// TIA Portal project "LinkedList_v000_000_004" (V16)
// task for 000.000.004: create LinkedList.FindID

(* hardware
DEVICE "S7-1200 station_1"  S7-1200 Station
   slot 0: "Rack_0"  S7-1200 Rack  Rack  V1.0
   slot 1: "PLC_1"  CPU 1212C DC/DC/DC  6ES7 212-1AE40-0XB0  V4.4
*)

// ===== PLC "PLC_1"  CPU 1212C DC/DC/DC =====

VAR_GLOBAL   // PLC tag table "Default tag table"
   "System_Byte" AT %MB1 : Byte;
   "FirstScan" AT %M1.0 : Bool;
   "DiagStatusUpdate" AT %M1.1 : Bool;
   "AlwaysTRUE" AT %M1.2 : Bool;
   "AlwaysFALSE" AT %M1.3 : Bool;
   "Clock_Byte" AT %MB0 : Byte;
   "Clock_10Hz" AT %M0.0 : Bool;
   "Clock_5Hz" AT %M0.1 : Bool;
   "Clock_2.5Hz" AT %M0.2 : Bool;
   "Clock_2Hz" AT %M0.3 : Bool;
   "Clock_1.25Hz" AT %M0.4 : Bool;
   "Clock_1Hz" AT %M0.5 : Bool;
   "Clock_0.625Hz" AT %M0.6 : Bool;
   "Clock_0.5Hz" AT %M0.7 : Bool;
END_VAR

TYPE "LinkedList.Node.Payload.UDT"
   STRUCT
      id : Char;
      status : String;
   END_STRUCT;
END_TYPE

TYPE "LinkedList.Node.UDT"
   STRUCT
      payload : "LinkedList.Node.Payload.UDT";
      pointer : DInt;
   END_STRUCT;
END_TYPE

TYPE "LinkedList.UDT"
   STRUCT
      head : DInt;
      list : Array[0..4] of "LinkedList.Node.UDT";
   END_STRUCT;
END_TYPE

TYPE "Validate.LinkedList.FindPointer.UDT"
   STRUCT
      request : Bool;
      needle : DInt;
      not_found : DInt;
      index : DInt;
   END_STRUCT;
END_TYPE

TYPE "Validate.LinkedList.FindPayload.UDT"
   STRUCT
      request : Bool;
      needle : "LinkedList.Node.Payload.UDT";
      not_found : DInt;
      tail_address : DInt;
      index : DInt;
   END_STRUCT;
END_TYPE

TYPE "Validate.LinkedList.FindID.UDT"
   STRUCT
      request : Bool;
      needle : Char;
      not_found : DInt;
      tail_address : DInt;
      index : DInt;
   END_STRUCT;
END_TYPE

DATA_BLOCK "LinkedList.IDB"   // DB1
{ S7_Optimized_Access := 'TRUE' }
AUTHOR : Machado
FAMILY : LinkedList
VERSION : 0.1
// stored: InstanceOfName LinkedList
"LinkedList"
BEGIN
END_DATA_BLOCK

DATA_BLOCK "ValidationSignals"   // DB2
{ S7_Optimized_Access := 'TRUE' }
VERSION : 0.1
   VAR
      FindPointer : "Validate.LinkedList.FindPointer.UDT";
      FindPayload : "Validate.LinkedList.FindPayload.UDT";
      FindID : "Validate.LinkedList.FindID.UDT";
   END_VAR
BEGIN
END_DATA_BLOCK

FUNCTION_BLOCK "LinkedList"   // FB1, SCL
TITLE = Linked List
{ S7_Optimized_Access := 'TRUE' }
AUTHOR : Machado
FAMILY : LinkedList
VERSION : 0.1
   VAR
      list : "LinkedList.UDT";
   END_VAR
BEGIN
END_FUNCTION_BLOCK

FUNCTION "LinkedList.FindPointer" : DInt   // FC1, SCL
TITLE = Find Node by Pointer In Linked List
{ S7_Optimized_Access := 'TRUE' }
AUTHOR : Machado
FAMILY : LinkedList
VERSION : 0.1
// returns not_found when not found.
// otherwise returs index of parent array where node with needle value as pointer.
   VAR_INPUT
      needle : DInt;
      not_found : DInt;   // value returned to user if needle not found
   END_VAR
   VAR_IN_OUT
      haystack : "LinkedList.UDT";
   END_VAR
   VAR_TEMP
      i : DInt;
      size : DInt;
   END_VAR
BEGIN
   REGION "GET SIZE"
       #size := UDINT_TO_DINT("LinkedList.Node[].CountOfElements"(#haystack.list));
   END_REGION


   REGION "SEARCH"
       FOR #i := 0 TO #size - 1 DO
           // no match
           IF #haystack.list[#i]."pointer" <> #needle THEN
               CONTINUE;
           END_IF;
           // match
           #"LinkedList.FindPointer" := #i;
           RETURN;
       END_FOR;
   END_REGION


   REGION "NOT FOUND"
       #"LinkedList.FindPointer" := #not_found;
       RETURN;
   END_REGION
END_FUNCTION

FUNCTION "LinkedList.Node[].CountOfElements" : UDInt   // FC2, SCL
TITLE = Count Of Elements of an Array of Linked List Nodes
{ S7_Optimized_Access := 'TRUE' }
AUTHOR : Machado
FAMILY : LinkedList
VERSION : 0.1
   VAR_INPUT
      list : Variant;
   END_VAR
BEGIN
   #"LinkedList.Node[].CountOfElements" := CountOfElements(#list);
   RETURN;
END_FUNCTION

FUNCTION "LinkedList.FindPayload" : DInt   // FC3, SCL
TITLE = Finde Node Index By Payload
{ S7_Optimized_Access := 'TRUE' }
AUTHOR : Machado
FAMILY : LinkedList
VERSION : 0.1
   VAR_INPUT
      needle : "LinkedList.Node.Payload.UDT";
      not_found : DInt;
      tail_address : DInt;
   END_VAR
   VAR_IN_OUT
      haystack : "LinkedList.UDT";
   END_VAR
   VAR_TEMP
      size : DInt;
      this_node : "LinkedList.Node.UDT";
      next_node : "LinkedList.Node.UDT";
      nodes_visited : DInt;
   END_VAR
BEGIN
   REGION "GET SIZE"
       #size := UDINT_TO_DINT("LinkedList.Node[].CountOfElements"(#haystack.list));
   END_REGION


   REGION "PRE-CONDITIONS"
       IF NOT "DInt.InRange"(x := #haystack.head, max := #size - 1, min := 0) THEN
           #"LinkedList.FindPayload" := #not_found;
           RETURN;
       END_IF;
   END_REGION


   REGION "PRIME WHILE LOOP"
       #this_node := #haystack.list[#haystack.head];
       IF #this_node.payload = #needle THEN
           #"LinkedList.FindPayload" := #haystack.head;
           RETURN;
       END_IF;
       #nodes_visited := 1;
   END_REGION


   REGION "SEARCH"
       WHILE #this_node."pointer" <> #tail_address DO
           #next_node := #haystack.list[#this_node."pointer"];
           IF #next_node.payload = #needle THEN
               #"LinkedList.FindPayload" := #this_node."pointer";
               RETURN;
           END_IF;
           #nodes_visited += 1;
           IF #nodes_visited > #size THEN
               #"LinkedList.FindPayload" := #not_found;
               RETURN;
           END_IF;
           #this_node := #next_node;
       END_WHILE;
   END_REGION


   REGION "NOT FOUND"
       #"LinkedList.FindPayload" := #not_found;
       RETURN;
   END_REGION
END_FUNCTION

FUNCTION "DInt.InRange" : Bool   // FC4, SCL
TITLE = Value Is In Range
{ S7_Optimized_Access := 'TRUE' }
AUTHOR : Machado
FAMILY : DInt
VERSION : 0.1
   VAR_INPUT
      x : DInt;
      max : DInt;
      min : DInt;
   END_VAR
BEGIN
   #"DInt.InRange" := #min <= #x AND #x <= #max;
END_FUNCTION

FUNCTION "LinkedList.FindID" : DInt   // FC5, SCL
TITLE = Finde Node Index By Payload
{ S7_Optimized_Access := 'TRUE' }
AUTHOR : Machado
FAMILY : LinkedList
VERSION : 0.1
   VAR_INPUT
      needle : Char;
      not_found : DInt;
      tail_address : DInt;
   END_VAR
   VAR_IN_OUT
      haystack : "LinkedList.UDT";
   END_VAR
   VAR_TEMP
      size : DInt;
      this_node : "LinkedList.Node.UDT";
      next_node : "LinkedList.Node.UDT";
      nodes_visited : DInt;
   END_VAR
BEGIN
   REGION "GET SIZE"
       #size := UDINT_TO_DINT("LinkedList.Node[].CountOfElements"(#haystack.list));
   END_REGION


   REGION "PRE-CONDITIONS"
       IF NOT "DInt.InRange"(x := #haystack.head, max := #size - 1, min := 0) THEN
           #"LinkedList.FindID" := #not_found;
           RETURN;
       END_IF;
   END_REGION


   REGION "PRIME WHILE LOOP"
       #this_node := #haystack.list[#haystack.head];
       IF #this_node.payload.id = #needle THEN
           #"LinkedList.FindID" := #haystack.head;
           RETURN;
       END_IF;
       #nodes_visited := 1;
   END_REGION


   REGION "SEARCH"
       WHILE #this_node."pointer" <> #tail_address DO
           #next_node := #haystack.list[#this_node."pointer"];
           IF #next_node.payload.id = #needle THEN
               #"LinkedList.FindID" := #this_node."pointer";
               RETURN;
           END_IF;
           #nodes_visited += 1;
           IF #nodes_visited > #size THEN
               #"LinkedList.FindID" := #not_found;
               RETURN;
           END_IF;
           #this_node := #next_node;
       END_WHILE;
   END_REGION


   REGION "NOT FOUND"
       #"LinkedList.FindID" := #not_found;
       RETURN;
   END_REGION
END_FUNCTION

ORGANIZATION_BLOCK "Main"   // OB1, LAD, ProgramCycle
TITLE = "Main Program Sweep (Cycle)"
{ S7_Optimized_Access := 'TRUE' }
VERSION : 0.1
   VAR_INPUT
      Initial_Call : Bool;   // Initial call of this OB
      Remanence : Bool;   // =True, if remanent data are available
   END_VAR
   VAR_TEMP   // added for the SCL form of the ladder/FBD networks
      _w1 : Bool;
   END_VAR
BEGIN

REGION Network 1: CALL LINKED LIST
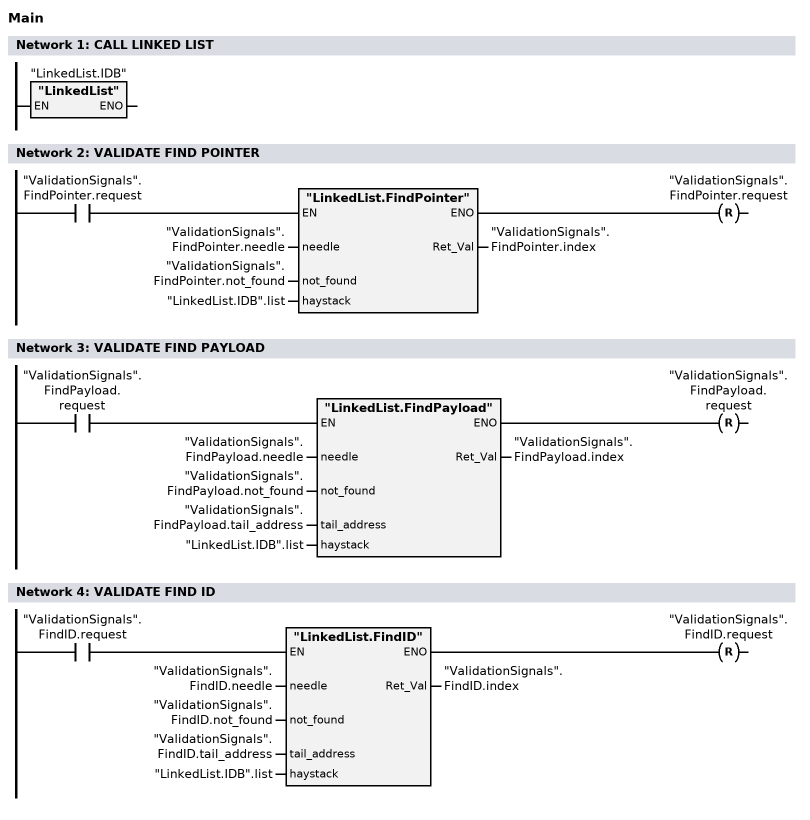
   RUNG wire#powerrail
      "LinkedList.IDB"()
   END_RUNG
   // the same network as SCL:
   "LinkedList.IDB"();   // "LinkedList"
END_REGION

REGION Network 2: VALIDATE FIND POINTER
   RUNG wire#powerrail
      Contact( "ValidationSignals".FindPointer.request )
      "LinkedList.FindPointer"(needle := "ValidationSignals".FindPointer.needle, not_found := "ValidationSignals".FindPointer.not_found, haystack := "LinkedList.IDB".list, Ret_Val => "ValidationSignals".FindPointer.index)
      R_Coil( "ValidationSignals".FindPointer.request )
   END_RUNG
   // the same network as SCL:
   "ValidationSignals".FindPointer.index := "LinkedList.FindPointer"(EN := "ValidationSignals".FindPointer.request,
                           needle := "ValidationSignals".FindPointer.needle,
                           not_found := "ValidationSignals".FindPointer.not_found,
                           haystack := "LinkedList.IDB".list,
                           ENO => #_w1);
   IF #_w1 THEN "ValidationSignals".FindPointer.request := FALSE; END_IF;
END_REGION

REGION Network 3: VALIDATE FIND PAYLOAD
   RUNG wire#powerrail
      Contact( "ValidationSignals".FindPayload.request )
      "LinkedList.FindPayload"(needle := "ValidationSignals".FindPayload.needle, not_found := "ValidationSignals".FindPayload.not_found, tail_address := "ValidationSignals".FindPayload.tail_address, haystack := "LinkedList.IDB".list, Ret_Val => "ValidationSignals".FindPayload.index)
      R_Coil( "ValidationSignals".FindPayload.request )
   END_RUNG
   // the same network as SCL:
   "ValidationSignals".FindPayload.index := "LinkedList.FindPayload"(EN := "ValidationSignals".FindPayload.request,
                           needle := "ValidationSignals".FindPayload.needle,
                           not_found := "ValidationSignals".FindPayload.not_found,
                           tail_address := "ValidationSignals".FindPayload.tail_address,
                           haystack := "LinkedList.IDB".list,
                           ENO => #_w1);
   IF #_w1 THEN "ValidationSignals".FindPayload.request := FALSE; END_IF;
END_REGION

REGION Network 4: VALIDATE FIND ID
   RUNG wire#powerrail
      Contact( "ValidationSignals".FindID.request )
      "LinkedList.FindID"(needle := "ValidationSignals".FindID.needle, not_found := "ValidationSignals".FindID.not_found, tail_address := "ValidationSignals".FindID.tail_address, haystack := "LinkedList.IDB".list, Ret_Val => "ValidationSignals".FindID.index)
      R_Coil( "ValidationSignals".FindID.request )
   END_RUNG
   // the same network as SCL:
   "ValidationSignals".FindID.index := "LinkedList.FindID"(EN := "ValidationSignals".FindID.request,
                           needle := "ValidationSignals".FindID.needle,
                           not_found := "ValidationSignals".FindID.not_found,
                           tail_address := "ValidationSignals".FindID.tail_address,
                           haystack := "LinkedList.IDB".list,
                           ENO => #_w1);
   IF #_w1 THEN "ValidationSignals".FindID.request := FALSE; END_IF;
END_REGION
END_ORGANIZATION_BLOCK